// TwinCAT 3 PLC project HMI_PLC
// ProgramVersion: 3.1.4024.0
// libraries:
//   State Machine Twincat, * (Home)
//   Tc2_Standard, * (Beckhoff Automation GmbH)
//   Tc2_System, * (Beckhoff Automation GmbH)
//   Tc3_JsonXml, * (Beckhoff Automation GmbH)
//   Tc3_Module, * (Beckhoff Automation GmbH)
//   VisuSymbols,3.5.10.0,System
// project tree:
//   DUTs/ ST_CameraStates.TcDUT
//   GVLs/ Hardware_Mapping.TcGVL, Cognex_Mapping.TcGVL
//   / PlcTask.TcTTO
//   POUs/ MAIN.TcPOU, _5000_PRG_Aborting.TcPOU, _1000_PRG_Homing.TcPOU, _3000_PRG_Running.TcPOU, _2000_PRG_Stopping.TcPOU, _4000_PRG_Pausing.TcPOU, _6000_PRG_Proceeding.TcPOU, VisualizationManager.TcVMO (not stored)
// real-time tasks:
//   TASK PlcTask: cycle T#10ms, priority 20, ADS port 350
//   TASK VISU_TASK: cycle T#200000us, priority 30, ADS port 351
//   TASK IO Task New: cycle T#1ms, priority 1, ADS port 301
// motion (NC):
//   TASK NC-Task 1 SAF: cycle T#2ms, priority 4, ADS port 501
//   TASK NC-Task 1 SVB: cycle T#10ms, priority 8, ADS port 511
//   AXIS Axis 1 (id 1)
//     OtherSettings: AllowMotionCmdToSlave=true
//     encoder EncType=4
//       EncPara: MaxCount=#x0000ffff
//         Inc: RefSoftSyncMask=#x0000ffff
//     drive DrvType=24
//       Analog: TorqueSetpointScale=10, ScaleFactorActTorque=0.1
//       TimeComp: TaskDelayCycles=1
//     controller CtrType=1
//       CtrPara: PriorControlFactor=1
//         Observer: BandWidth=20
//   AXIS Axis 2 (id 2)
//     OtherSettings: AllowMotionCmdToSlave=true
//     encoder EncType=4
//       EncPara: MaxCount=#x0000ffff
//         Inc: RefSoftSyncMask=#x0000ffff
//     drive DrvType=24
//       Analog: TorqueSetpointScale=10, ScaleFactorActTorque=0.1
//       TimeComp: TaskDelayCycles=1
//     controller CtrType=1
//       CtrPara: PriorControlFactor=1
//         Observer: BandWidth=20
// I/O:
//   DEVICE Device 1 (TC3 EIP Scanner), AmsNetId 172.18.236.100.2.1
//     Box 1 (In-Sight 7000 Series) // <INFO> </INFO> <EDS> C:\TwinCAT\3.1\Config\Io\EtherNetIP\02A6006401090C00.eds </EDS>
//   DEVICE Device 2 (EtherCAT), AmsNetId 172.18.236.100.3.1
//     Term 2 (EK1100) [EK1100 EtherCAT Coupler (2A E-Bus)]
//       Term 3 (EL1008) [EL1008 8Ch. Dig. Input 24V, 3ms]
//       Term 4 (EL1008) [EL1008 8Ch. Dig. Input 24V, 3ms]
//       Term 5 (EL2008) [EL2008 8Ch. Dig. Output 24V, 0.5A]
//       Term 6 (EL2008) [EL2008 8Ch. Dig. Output 24V, 0.5A]
//       Term 7 (EL7047) [EL7047 1Ch. Stepper motor output stage (50V, 5A)]
//       Term 8 (EL7047) [EL7047 1Ch. Stepper motor output stage (50V, 5A)]
//       Term 8 (EL9011) [EL9011 End Terminal]
// variable links:
//   NC-Task 1 SAF/Axes/Axis 1 <-> Device 2 (EtherCAT)/Term 2 (EK1100)/Term 7 (EL7047)
//     Drive/Inputs/In/nState1 @bit 3 <-> STM Status/Status/Error
//     Drive/Inputs/In/nState1 @bit 7 <-> STM Status/Status/Motor stall
//     Drive/Inputs/In/nState1 @bit 5 <-> STM Status/Status/Moving negative
//     Drive/Inputs/In/nState1 @bit 4 <-> STM Status/Status/Moving positive
//     Drive/Inputs/In/nState1 @bit 1 <-> STM Status/Status/Ready
//     Drive/Inputs/In/nState1 <-> STM Status/Status/Ready to enable
//     Drive/Inputs/In/nState1 @bit 6 <-> STM Status/Status/Torque reduced
//     Drive/Inputs/In/nState1 @bit 2 <-> STM Status/Status/Warning
//     Drive/Inputs/In/nState2 @bit 3 <-> STM Status/Status/Digital input 1
//     Drive/Inputs/In/nState2 @bit 4 <-> STM Status/Status/Digital input 2
//     Drive/Inputs/In/nState2 @bit 5 <-> STM Status/Status/Sync error
//     Drive/Inputs/In/nState2 @bit 7 <-> STM Status/Status/TxPDO Toggle
//     Drive/Inputs/In/nState4 @bit 1 <-> WcState/InputToggle
//     Drive/Inputs/In/nState4 <-> WcState/WcState
//     Drive/Outputs/Out/nCtrl1 <-> STM Control/Control/Enable
//     Drive/Outputs/Out/nCtrl1 @bit 2 <-> STM Control/Control/Reduce torque
//     Drive/Outputs/Out/nCtrl1 @bit 1 <-> STM Control/Control/Reset
//     Drive/Outputs/Out/nCtrl2 @bit 3 <-> STM Control/Control/Digital output 1
//     Drive/Outputs/Out/nDataOut2[0] <-> STM Velocity/Velocity
//     Enc/Inputs/In/nDataIn1[0] <-> ENC Status compact/Counter value
//     Enc/Inputs/In/nDataIn2[0] <-> ENC Status compact/Latch value
//     Enc/Inputs/In/nState1 @bit 4 <-> ENC Status compact/Status/Counter overflow
//     Enc/Inputs/In/nState1 @bit 3 <-> ENC Status compact/Status/Counter underflow
//     Enc/Inputs/In/nState1 @bit 7 <-> ENC Status compact/Status/Extrapolation stall
//     Enc/Inputs/In/nState1 <-> ENC Status compact/Status/Latch C valid
//     Enc/Inputs/In/nState1 @bit 1 <-> ENC Status compact/Status/Latch extern valid
//     Enc/Inputs/In/nState1 @bit 2 <-> ENC Status compact/Status/Set counter done
//     Enc/Inputs/In/nState2 @bit 4 <-> ENC Status compact/Status/Status of extern latch
//     Enc/Inputs/In/nState2 <-> ENC Status compact/Status/Status of input A
//     Enc/Inputs/In/nState2 @bit 1 <-> ENC Status compact/Status/Status of input B
//     Enc/Inputs/In/nState2 @bit 2 <-> ENC Status compact/Status/Status of input C
//     Enc/Inputs/In/nState2 @bit 5 <-> ENC Status compact/Status/Sync error
//     Enc/Inputs/In/nState2 @bit 7 <-> ENC Status compact/Status/TxPDO Toggle
//     Enc/Inputs/In/nState4 @bit 1 <-> WcState/InputToggle
//     Enc/Inputs/In/nState4 <-> WcState/WcState
//     Enc/Outputs/Out/nCtrl1 <-> ENC Control compact/Control/Enable latch C
//     Enc/Outputs/Out/nCtrl1 @bit 3 <-> ENC Control compact/Control/Enable latch extern on negative edge
//     Enc/Outputs/Out/nCtrl1 @bit 1 <-> ENC Control compact/Control/Enable latch extern on positive edge
//     Enc/Outputs/Out/nCtrl1 @bit 2 <-> ENC Control compact/Control/Set counter
//     Enc/Outputs/Out/nDataOut1[0] <-> ENC Control compact/Set counter value
//   NC-Task 1 SAF/Axes/Axis 2 <-> Device 2 (EtherCAT)/Term 2 (EK1100)/Term 8 (EL7047)
//     Drive/Inputs/In/nState1 @bit 3 <-> STM Status/Status/Error
//     Drive/Inputs/In/nState1 @bit 7 <-> STM Status/Status/Motor stall
//     Drive/Inputs/In/nState1 @bit 5 <-> STM Status/Status/Moving negative
//     Drive/Inputs/In/nState1 @bit 4 <-> STM Status/Status/Moving positive
//     Drive/Inputs/In/nState1 @bit 1 <-> STM Status/Status/Ready
//     Drive/Inputs/In/nState1 <-> STM Status/Status/Ready to enable
//     Drive/Inputs/In/nState1 @bit 6 <-> STM Status/Status/Torque reduced
//     Drive/Inputs/In/nState1 @bit 2 <-> STM Status/Status/Warning
//     Drive/Inputs/In/nState2 @bit 3 <-> STM Status/Status/Digital input 1
//     Drive/Inputs/In/nState2 @bit 4 <-> STM Status/Status/Digital input 2
//     Drive/Inputs/In/nState2 @bit 5 <-> STM Status/Status/Sync error
//     Drive/Inputs/In/nState2 @bit 7 <-> STM Status/Status/TxPDO Toggle
//     Drive/Inputs/In/nState4 @bit 1 <-> WcState/InputToggle
//     Drive/Inputs/In/nState4 <-> WcState/WcState
//     Drive/Outputs/Out/nCtrl1 <-> STM Control/Control/Enable
//     Drive/Outputs/Out/nCtrl1 @bit 2 <-> STM Control/Control/Reduce torque
//     Drive/Outputs/Out/nCtrl1 @bit 1 <-> STM Control/Control/Reset
//     Drive/Outputs/Out/nCtrl2 @bit 3 <-> STM Control/Control/Digital output 1
//     Drive/Outputs/Out/nDataOut2[0] <-> STM Velocity/Velocity
//     Enc/Inputs/In/nDataIn1[0] <-> ENC Status compact/Counter value
//     Enc/Inputs/In/nDataIn2[0] <-> ENC Status compact/Latch value
//     Enc/Inputs/In/nState1 @bit 4 <-> ENC Status compact/Status/Counter overflow
//     Enc/Inputs/In/nState1 @bit 3 <-> ENC Status compact/Status/Counter underflow
//     Enc/Inputs/In/nState1 @bit 7 <-> ENC Status compact/Status/Extrapolation stall
//     Enc/Inputs/In/nState1 <-> ENC Status compact/Status/Latch C valid
//     Enc/Inputs/In/nState1 @bit 1 <-> ENC Status compact/Status/Latch extern valid
//     Enc/Inputs/In/nState1 @bit 2 <-> ENC Status compact/Status/Set counter done
//     Enc/Inputs/In/nState2 @bit 4 <-> ENC Status compact/Status/Status of extern latch
//     Enc/Inputs/In/nState2 <-> ENC Status compact/Status/Status of input A
//     Enc/Inputs/In/nState2 @bit 1 <-> ENC Status compact/Status/Status of input B
//     Enc/Inputs/In/nState2 @bit 2 <-> ENC Status compact/Status/Status of input C
//     Enc/Inputs/In/nState2 @bit 5 <-> ENC Status compact/Status/Sync error
//     Enc/Inputs/In/nState2 @bit 7 <-> ENC Status compact/Status/TxPDO Toggle
//     Enc/Inputs/In/nState4 @bit 1 <-> WcState/InputToggle
//     Enc/Inputs/In/nState4 <-> WcState/WcState
//     Enc/Outputs/Out/nCtrl1 <-> ENC Control compact/Control/Enable latch C
//     Enc/Outputs/Out/nCtrl1 @bit 3 <-> ENC Control compact/Control/Enable latch extern on negative edge
//     Enc/Outputs/Out/nCtrl1 @bit 1 <-> ENC Control compact/Control/Enable latch extern on positive edge
//     Enc/Outputs/Out/nCtrl1 @bit 2 <-> ENC Control compact/Control/Set counter
//     Enc/Outputs/Out/nDataOut1[0] <-> ENC Control compact/Set counter value
//   HMI-PLC/HMI-PLC Instance <-> Device 1 (TC3 EIP Scanner)/Box 1 (In-Sight 7000 Series)
//     PlcTask Inputs/IO_Mapping.inpAcquiring <-> Connection 1 (Input/Output)/Inputs/Acquiring
//     PlcTask Inputs/IO_Mapping.inpAcquisitionID <-> Connection 1 (Input/Output)/Inputs/Acquisition ID
//     PlcTask Inputs/IO_Mapping.inpCommandComplete <-> Connection 1 (Input/Output)/Inputs/Command Complete
//     PlcTask Inputs/IO_Mapping.inpCommandExecuting <-> Connection 1 (Input/Output)/Inputs/Command Executing
//     PlcTask Inputs/IO_Mapping.inpCommandFailed <-> Connection 1 (Input/Output)/Inputs/Command Failed
//     PlcTask Inputs/IO_Mapping.inpCurrentJobID <-> Connection 1 (Input/Output)/Inputs/Current Job ID
//     PlcTask Inputs/IO_Mapping.inpExposureComplete <-> Connection 1 (Input/Output)/Inputs/Exposure Complete
//     PlcTask Inputs/IO_Mapping.inpInspecting <-> Connection 1 (Input/Output)/Inputs/Inspecting
//     PlcTask Inputs/IO_Mapping.inpInspectionComplete <-> Connection 1 (Input/Output)/Inputs/Inspection Complete
//     PlcTask Inputs/IO_Mapping.inpInspectionID <-> Connection 1 (Input/Output)/Inputs/Inspection ID
//     PlcTask Inputs/IO_Mapping.inpInspectionResultCode <-> Connection 1 (Input/Output)/Inputs/Inspection Result Code
//     PlcTask Inputs/IO_Mapping.inpInspectionResults <-> Connection 1 (Input/Output)/Inputs/Inspection Results
//     PlcTask Inputs/IO_Mapping.inpInspectionResults{1..10} <-> Connection 1 (Input/Output)/Inputs/Inspection Results_{1..10}  (10 links)
//     PlcTask Inputs/IO_Mapping.inpJobPass <-> Connection 1 (Input/Output)/Inputs/Job Pass
//     PlcTask Inputs/IO_Mapping.inpMissedAcq <-> Connection 1 (Input/Output)/Inputs/Missed Acq
//     PlcTask Inputs/IO_Mapping.inpOfflineReason <-> Connection 1 (Input/Output)/Inputs/Offline Reason
//     PlcTask Inputs/IO_Mapping.inpOnline <-> Connection 1 (Input/Output)/Inputs/Online
//     PlcTask Inputs/IO_Mapping.inpResultsBufferOverrun <-> Connection 1 (Input/Output)/Inputs/Results Buffer Overrun
//     PlcTask Inputs/IO_Mapping.inpResultsValid <-> Connection 1 (Input/Output)/Inputs/Results Valid
//     PlcTask Inputs/IO_Mapping.inpTestRunReady <-> Connection 1 (Input/Output)/Inputs/Test Run Ready
//     PlcTask Inputs/IO_Mapping.inpTriggerAck <-> Connection 1 (Input/Output)/Inputs/Trigger Ack
//     PlcTask Inputs/IO_Mapping.inpTriggerReady <-> Connection 1 (Input/Output)/Inputs/Trigger Ready
//     PlcTask Outputs/IO_Mapping.outBufferResultsEnable <-> Connection 1 (Input/Output)/Outputs/Buffer Results Enable
//     PlcTask Outputs/IO_Mapping.outCommand <-> Connection 1 (Input/Output)/Outputs/Command
//     PlcTask Outputs/IO_Mapping.outExecuteCommand <-> Connection 1 (Input/Output)/Outputs/Execute Command
//     PlcTask Outputs/IO_Mapping.outInspectionResultsAck <-> Connection 1 (Input/Output)/Outputs/Inspection Results Ack
//     PlcTask Outputs/IO_Mapping.outSetOffline <-> Connection 1 (Input/Output)/Outputs/Set Offline
//     PlcTask Outputs/IO_Mapping.outSoftEvent{0..7} <-> Connection 1 (Input/Output)/Outputs/Soft Event {0..7}  (8 links)
//     PlcTask Outputs/IO_Mapping.outTriggerCamera <-> Connection 1 (Input/Output)/Outputs/Trigger
//     PlcTask Outputs/IO_Mapping.outTriggerEnable <-> Connection 1 (Input/Output)/Outputs/Trigger Enable
//     PlcTask Outputs/IO_Mapping.outUserData <-> Connection 1 (Input/Output)/Outputs/User Data
//     PlcTask Outputs/IO_Mapping.outUserData{1..10} <-> Connection 1 (Input/Output)/Outputs/User Data_{1..10}  (10 links)
//   HMI-PLC/HMI-PLC Instance <-> Device 2 (EtherCAT)/Term 2 (EK1100)/Term 3 (EL1008)
//     PlcTask Inputs/IO_Mapping.input1 <-> Channel 1/Input
//     PlcTask Inputs/IO_Mapping.input2 <-> Channel 2/Input
//   HMI-PLC/HMI-PLC Instance <-> Device 2 (EtherCAT)/Term 2 (EK1100)/Term 5 (EL2008)
//     PlcTask Outputs/IO_Mapping.output1 <-> Channel 1/Output
//     PlcTask Outputs/IO_Mapping.output2 <-> Channel 2/Output

CONFIGURATION HMI_PLC
    RESOURCE PLC ON TwinCAT3
        TASK PlcTask(INTERVAL := T#10ms, PRIORITY := 20);
        PROGRAM MAIN WITH PlcTask : MAIN;
    END_RESOURCE
END_CONFIGURATION

// ---- DUTs/ST_CameraStates.TcDUT
TYPE ST_CameraState :
STRUCT
    stsIdle              : BOOL := FALSE;
    stsReadyToTrigger    : BOOL := FALSE;
    stsTriggering        : BOOL := FALSE;
    stsAcquiring         : BOOL := FALSE;
    stsWaitResults       : BOOL := FALSE;
    stsProcessResults    : BOOL := FALSE;
    stsError             : BOOL := FALSE;
END_STRUCT
END_TYPE

// ---- GVLs/Hardware_Mapping.TcGVL
{attribute 'qualified_only'}
VAR_GLOBAL
END_VAR

// ---- GVLs/Cognex_Mapping.TcGVL
{attribute 'qualified_only'}
VAR_GLOBAL
	
	// COGNEX INSIGHT 7000 EIP EDS MAPPING
	//--------------------------------------
	// Inputs
	inpTriggerReady AT %I* : BOOL;
	inpTriggerAck AT %I* : BOOL;
	inpAcquiring AT %I* : BOOL;
	inpMissedAcq AT %I* : BOOL;
	inpOfflineReason AT %I* : USINT; // 3 bits represented as USINT (8 bits)
	inpOnline AT %I* : BOOL;
	inpInspecting AT %I* : BOOL;
	inpInspectionComplete AT %I* : BOOL;
	inpResultsBufferOverrun AT %I* : BOOL;
	inpResultsValid AT %I* : BOOL;
	inpCommandExecuting AT %I* : BOOL;
	inpCommandComplete AT %I* : BOOL;
	inpCommandFailed AT %I* : BOOL;
	inpNoname0ArrBIT AT %I* : ARRAY[0..1] OF BOOL;
	inpExposureComplete AT %I* : BOOL;
	inpJobPass AT %I* : BOOL;
	inpTestRunReady AT %I* : BOOL;
	inpNoname1ArrBIT AT %I* : ARRAY[0..1] OF BOOL;
	inpCurrentJobID AT %I* : UINT;
	inpAcquisitionID AT %I* : UINT;
	inpInspectionID AT %I* : UINT;
	inpInspectionResultCode AT %I* : INT;
	inpInspectionResults AT %I* : BYTE;
	inpInspectionResults1 AT %I* : BYTE;
	inpInspectionResults2 AT %I* : BYTE;
	inpInspectionResults3 AT %I* : BYTE;
	inpInspectionResults4 AT %I* : BYTE;
	inpInspectionResults5 AT %I* : BYTE;
	inpInspectionResults6 AT %I* : BYTE;
	inpInspectionResults7 AT %I* : BYTE;
	inpInspectionResults8 AT %I* : BYTE;
	inpInspectionResults9 AT %I* : BYTE;
	inpInspectionResults10 AT %I* : BYTE;
	
	// Outputs
	outTriggerEnable AT %Q* : BOOL;
	outTriggerCamera AT %Q* : BOOL;
	outBufferResultsEnable AT %Q* : BOOL;
	outInspectionResultsAck AT %Q* : BOOL;
	outExecuteCommand AT %Q* : BOOL;
	outNoname0ArrBIT AT %Q* : ARRAY[0..1] OF BOOL;
	outSetOffline AT %Q* : BOOL;
	outSoftEvent0 AT %Q* : BOOL;
	outSoftEvent1 AT %Q* : BOOL;
	outSoftEvent2 AT %Q* : BOOL;
	outSoftEvent3 AT %Q* : BOOL;
	outSoftEvent4 AT %Q* : BOOL;
	outSoftEvent5 AT %Q* : BOOL;
	outSoftEvent6 AT %Q* : BOOL;
	outSoftEvent7 AT %Q* : BOOL;
	outCommand AT %Q* : UINT;
	outUserData AT %Q* : BYTE;
	outUserData1 AT %Q* : BYTE;
	outUserData2 AT %Q* : BYTE;
	outUserData3 AT %Q* : BYTE;
	outUserData4 AT %Q* : BYTE;
	outUserData5 AT %Q* : BYTE;
	outUserData6 AT %Q* : BYTE;
	outUserData7 AT %Q* : BYTE;
	outUserData8 AT %Q* : BYTE;
	outUserData9 AT %Q* : BYTE;
	outUserData10 AT %Q* : BYTE;
	//--------------------------------------
	
	
	// Regular IO 
	input1 AT %I* : BOOL;
	input2 AT %I* : BOOL;
	
	output1 AT %Q* : BOOL;
	output2 AT %Q* : BOOL;

END_VAR

// ---- POUs/MAIN.TcPOU
PROGRAM MAIN
VAR
    // State Machine instance
    fbStateMachine : FB_StateMachine;
    
    // HMI interface for state machine
    stateMachineHMI : SM_HMI;
    
    // Current step for state machine - SHARED between state machine and all step programs
    currentStep : ActiveStep;
    
    // State machine command inputs
    smCommands : ST_SM_Commands;
      
    // Test inputs for permissions
    testAutoIntlk : INT := -1;  // All OK by default (-1 = all bits OK)
    testHomePerm : INT := -1;   // All OK by default
    testStartPerm : INT := -1;  // All OK by default
    testProceedPerm : INT := -1; // All OK by default 

	NextStep: DINT; // Next step to be modified by sequences
	
END_VAR

//=============================================================================
// MAIN PROGRAM - State Machine Implementation with Sequence Programs
//=============================================================================

//=============================================================================
// CENTRALIZED INITIAL STEP SETTING
//=============================================================================
// Initialize sequence when first entering any state (CurrentStep.Step = 0)
IF currentStep.Step = 0 THEN
    IF fbStateMachine.Status.Homing THEN
        NextStep := 1000;  // Start homing sequence
        // Force immediate timer reset on state entry
        smCommands.CompleteState := FALSE;
    ELSIF fbStateMachine.Status.Running THEN
        NextStep := 3000;  // Start running sequence
        smCommands.CompleteState := FALSE;
    ELSIF fbStateMachine.Status.Stopping THEN
        NextStep := 2000;  // Start stopping sequence
        smCommands.CompleteState := FALSE;
    ELSIF fbStateMachine.Status.Aborting THEN
        NextStep := 5000;  // Start aborting sequence
        smCommands.CompleteState := FALSE;
    ELSIF fbStateMachine.Status.Pausing THEN
        NextStep := 4000;  // Start pausing sequence
        smCommands.CompleteState := FALSE;
    ELSIF fbStateMachine.Status.Proceeding THEN
        NextStep := 6000;  // Start proceeding sequence
        smCommands.CompleteState := FALSE;
    ELSE
        // No initial step needed
    END_IF;
END_IF;

// Call state machine BEFORE sequences to ensure timer is updated first
fbStateMachine(
    EnableIn := TRUE,              // Enable the state machine
    cfgAutoRun := TRUE,           // Auto run configuration  
    inpAutoIntlk := testAutoIntlk, // Auto interlocks
    inpHomePerm := testHomePerm,   // Home permissions
    inpStartPerm := testStartPerm, // Start permissions
    inpProceedPerm := testProceedPerm, // Proceed permissions
    NextStep := NextStep,  // Next step from active sequence program
    Commands := smCommands,        // Command inputs
    HMI := stateMachineHMI,        // HMI interface
    CurrentStep := currentStep     // Current step (shared with sequences)
);


//=============================================================================
// ALWAYS CALL ALL SEQUENCE PROGRAMS - AFTER STATE MACHINE
//=============================================================================
// This ensures the timer has been properly updated before sequences evaluate
// Call all sequence programs - FB_SequenceStep logic handles which steps are active
// This ensures all tags update in real-time for better HMI visibility
_1000_PRG_Homing(
    CurrentStep := currentStep,
    StepTimerSeconds := REAL_TO_DINT(fbStateMachine.StepInfo.StepTimerSeconds),
    RetrySignal := fbStateMachine.outRetry,
    StateMachineStatus := fbStateMachine.Status,
    NextStep := NextStep
);

_3000_PRG_Running(
    CurrentStep := currentStep,
    StepTimerSeconds := REAL_TO_DINT(fbStateMachine.StepInfo.StepTimerSeconds),
    RetrySignal := fbStateMachine.outRetry,
    StateMachineStatus := fbStateMachine.Status,
    NextStep := NextStep
);

_2000_PRG_Stopping(
    CurrentStep := currentStep,
    StepTimerSeconds := REAL_TO_DINT(fbStateMachine.StepInfo.StepTimerSeconds),
    RetrySignal := fbStateMachine.outRetry,
    StateMachineStatus := fbStateMachine.Status,
    NextStep := NextStep
);

_5000_PRG_Aborting(
    CurrentStep := currentStep,
    StepTimerSeconds := REAL_TO_DINT(fbStateMachine.StepInfo.StepTimerSeconds),
    RetrySignal := fbStateMachine.outRetry,
    StateMachineStatus := fbStateMachine.Status,
    NextStep := NextStep
);

_4000_PRG_Pausing(
    CurrentStep := currentStep,
    StepTimerSeconds := REAL_TO_DINT(fbStateMachine.StepInfo.StepTimerSeconds),
    RetrySignal := fbStateMachine.outRetry,
    StateMachineStatus := fbStateMachine.Status,
    NextStep := NextStep
);

_6000_PRG_Proceeding(
    CurrentStep := currentStep,
    StepTimerSeconds := REAL_TO_DINT(fbStateMachine.StepInfo.StepTimerSeconds),
    RetrySignal := fbStateMachine.outRetry,
    StateMachineStatus := fbStateMachine.Status,
    NextStep := NextStep
);

END_PROGRAM

// ---- POUs/_1000_PRG_Homing.TcPOU
PROGRAM _1000_PRG_Homing
VAR_IN_OUT
    CurrentStep : ActiveStep;  // Shared step structure with state machine
	NextStep: DINT; // Next step to be modified by sequences
END_VAR

VAR_INPUT
    StepTimerSeconds : DINT;   // Timer value from state machine
    RetrySignal : BOOL;        // Retry signal from state machine
    StateMachineStatus : ST_SM_Status;  // Complete state machine status
END_VAR


VAR
    // Step function blocks for homing sequence
    fbStep1000 : FB_SequenceStep;  // Home Initialize
    fbStep1002 : FB_SequenceStep;  // Home Execute
    
    // Step permissives (simulation for testing)
    step1000Perms : INT := -1;     // All OK for step 1000
    step1002Perms : INT := -1;     // All OK for step 1002
    
END_VAR

//=============================================================================
// PRG_Homing - Handles HOMING state sequence (1000-1999)
//=============================================================================
// Step numbering: 1000, 1002 (even numbers)
// Fault steps: 1001, 1003 (odd numbers, +1 of original)
// NOTE: Initial step setting (CurrentStep.Step = 0) is handled in MAIN program


//=============================================================================
// STEP 1000 - HOME INITIALIZE
//=============================================================================
fbStep1000(
    inpStep := CurrentStep.Step,
    cfgStep := 1000,
    cfgNextStep := 1002,
    inpStepTimerSeconds := StepTimerSeconds,
    inpRetry := RetrySignal,
    inpStepPermissives := step1000Perms,
    cfgStepTimeout := 10,  // 10 second timeout
    inpFaultStep := FALSE,
    ActiveStep := CurrentStep
);

// Step 1000 Active Logic
IF fbStep1000.outStepActive THEN
    // Only simulate permissives if step is active but not advancing
    IF fbStep1000.outNextStep = fbStep1000.cfgStep THEN  // Step is waiting for permissives
        // Permissives simulation - Simulate based on timer
        IF StepTimerSeconds < 3 THEN
            step1000Perms := 16#FFFE;  // Bit 0 not OK (not ready yet)
        ELSE
            step1000Perms := -1;  // All permissives OK after 3 seconds
        END_IF;
    END_IF;
    
    // HMI configuration and actions
    CurrentStep.PermsHMI.Name := 'Home Initialize';
    CurrentStep.PermsHMI.Desc[0] := 'System Ready';
    CurrentStep.PermsHMI.Desc[1] := 'Home Position Clear';
    CurrentStep.PermsHMI.Desc[2] := 'Safety Systems OK';
    
    // Add any step-specific actions here
    // Example: Reset position counters, check home sensors, etc.
    
    // FB_SequenceStep determines next step automatically based on permissives
    NextStep := fbStep1000.outNextStep;
ELSE
    // Reset permissives when step is not active (ensures fresh start next time)
    step1000Perms := 16#FFFE;  // Reset to NOT OK when leaving step
END_IF;

//=============================================================================
// STEP 1002 - HOME EXECUTE
//=============================================================================
fbStep1002(
    inpStep := CurrentStep.Step,
    cfgStep := 1002,
    cfgNextStep := 0,  // sequence complete
    inpStepTimerSeconds := StepTimerSeconds,
    inpRetry := RetrySignal,
    inpStepPermissives := step1002Perms,
    cfgStepTimeout := 15,  // 15 second timeout
    inpFaultStep := FALSE,
    ActiveStep := CurrentStep
);

// Step 1002 Active Logic
IF fbStep1002.outStepActive THEN
    // Only simulate permissives if step is active but not advancing
    IF fbStep1002.outNextStep = fbStep1002.cfgStep THEN  // Step is waiting for permissives
        // Permissives simulation - Simulate based on timer
        IF StepTimerSeconds < 8 THEN
            step1002Perms := 16#FFFD;  // Bit 1 not OK (homing not complete)
        ELSE
            step1002Perms := -1;  // All permissives OK after 8 seconds
        END_IF;
    END_IF;
    
    // HMI configuration and actions
    CurrentStep.PermsHMI.Name := 'Home Execute';
    CurrentStep.PermsHMI.Desc[0] := 'Motors Enabled';
    CurrentStep.PermsHMI.Desc[1] := 'Home Sensors Active';
    CurrentStep.PermsHMI.Desc[2] := 'No Emergency Stops';
    
    // Add any step-specific actions here
    // Example: Start homing motion, monitor position feedback, etc.
    
    // FB_SequenceStep determines next step automatically based on permissives
    NextStep := fbStep1002.outNextStep;
ELSE
    // Reset permissives when step is not active (ensures fresh start next time)
    step1002Perms := 16#FFFD;  // Reset to NOT OK when leaving step
END_IF;

END_PROGRAM

// ---- POUs/_3000_PRG_Running.TcPOU
PROGRAM _3000_PRG_Running
VAR_IN_OUT
    CurrentStep : ActiveStep;  // Shared step structure with state machine
	NextStep: DINT; // Next step to be modified by sequences
END_VAR
VAR_INPUT
    StepTimerSeconds : DINT;   // Timer value from state machine
    RetrySignal : BOOL;        // Retry signal from state machine
    StateMachineStatus : ST_SM_Status;  // Complete state machine status
END_VAR

VAR
    // Step function blocks for running sequence
    fbStep3000 : FB_SequenceStep;  // Production Start
    fbStep3002 : FB_SequenceStep;  // Production Execute
    fbStep3004 : FB_SequenceStep;  // Production Quality Check
    fbStep3006 : FB_SequenceStep;  // Packaging Prepare
    fbStep3008 : FB_SequenceStep;  // Production Finalize
    
    // Step permissives (simulation for testing)
    step3000Perms : INT := -1;     // All OK for step 3000
    step3002Perms : INT := -1;     // All OK for step 3002
    step3004Perms : INT := -1;     // All OK for step 3004
    step3006Perms : INT := -1;     // All OK for step 3006
    step3008Perms : INT := -1;     // All OK for step 3008
    
END_VAR

//=============================================================================
// PRG_Running - Handles RUNNING state sequence (3000-3999)
//=============================================================================
// Step numbering: 3000, 3002 (even numbers)
// Fault steps: 3001, 3003 (odd numbers, +1 of original)
// NOTE: Initial step setting (CurrentStep.Step = 0) is handled in MAIN program


//=============================================================================
// STEP 3000 - PRODUCTION START
//=============================================================================
fbStep3000(
    inpStep := CurrentStep.Step,
    cfgStep := 3000,
    cfgNextStep := 3002,
    inpStepTimerSeconds := StepTimerSeconds,
    inpRetry := RetrySignal,
    inpStepPermissives := step3000Perms,
    cfgStepTimeout := 12,  // 12 second timeout
    inpFaultStep := FALSE,
    ActiveStep := CurrentStep
);

// Step 3000 Active Logic
IF fbStep3000.outStepActive THEN
    // Only simulate permissives if step is active but not advancing
    IF fbStep3000.outNextStep = fbStep3000.cfgStep THEN  // Step is waiting for permissives
        // Permissives simulation - Simulate based on timer
        IF StepTimerSeconds < 3 THEN
            step3000Perms := 16#FFFE;  // Bit 0 not OK (not ready yet)
        ELSE
            step3000Perms := -1;  // All permissives OK after 5 seconds
        END_IF;
    END_IF;
    
    // HMI configuration and actions
    CurrentStep.PermsHMI.Name := 'Production Start';
    CurrentStep.PermsHMI.Desc[0] := 'Raw Material Available';
    CurrentStep.PermsHMI.Desc[1] := 'Process Temperature OK';
    CurrentStep.PermsHMI.Desc[2] := 'Quality System Ready';
    
    // Add any step-specific actions here
    // Example: Start production line, initialize process parameters, etc.
    
    // FB_SequenceStep determines next step automatically based on permissives
    NextStep := fbStep3000.outNextStep;
ELSE
    // Reset permissives when step is not active (ensures fresh start next time)
    step3000Perms := 16#FFFE;  // Reset to NOT OK when leaving step
END_IF;

//=============================================================================
// STEP 3002 - PRODUCTION EXECUTE
//=============================================================================
fbStep3002(
    inpStep := CurrentStep.Step,
    cfgStep := 3002,
    cfgNextStep := 3004,
    inpStepTimerSeconds := StepTimerSeconds,
    inpRetry := RetrySignal,
    inpStepPermissives := step3002Perms,
    cfgStepTimeout := 20,  // 20 second timeout
    inpFaultStep := FALSE,
    ActiveStep := CurrentStep
);

// Step 3002 Active Logic
IF fbStep3002.outStepActive THEN
    // Only simulate permissives if step is active but not advancing
    IF fbStep3002.outNextStep = fbStep3002.cfgStep THEN  // Step is waiting for permissives
        // Permissives simulation - Simulate based on timer
        IF StepTimerSeconds < 4 THEN
            step3002Perms := 16#FFFD;  // Bit 1 not OK (production not complete)
        ELSE
            step3002Perms := -1;  // All permissives OK after 15 seconds
        END_IF;
    END_IF;
    
    // HMI configuration and actions
    CurrentStep.PermsHMI.Name := 'Production Execute';
    CurrentStep.PermsHMI.Desc[0] := 'Production Line Running';
    CurrentStep.PermsHMI.Desc[1] := 'Quality Checks Passing';
    CurrentStep.PermsHMI.Desc[2] := 'Output Quality OK';
    
    // Add any step-specific actions here
    // Example: Monitor production process, quality checks, output control, etc.
    
    // FB_SequenceStep determines next step automatically based on permissives
    NextStep := fbStep3002.outNextStep;
ELSE
    // Reset permissives when step is not active (ensures fresh start next time)
    step3002Perms := 16#FFFD;  // Reset to NOT OK when leaving step
END_IF;

//=============================================================================
// STEP 3004 - PRODUCTION QUALITY CHECK
//=============================================================================
fbStep3004(
    inpStep := CurrentStep.Step,
    cfgStep := 3004,
    cfgNextStep := 3006,
    inpStepTimerSeconds := StepTimerSeconds,
    inpRetry := RetrySignal,
    inpStepPermissives := step3004Perms,
    cfgStepTimeout := 12,  // 12 second timeout
    inpFaultStep := FALSE,
    ActiveStep := CurrentStep
);

IF fbStep3004.outStepActive THEN
    // Only simulate permissives if step is active but not advancing
    IF fbStep3004.outNextStep = fbStep3004.cfgStep THEN  // Step is waiting for permissives
        // Simulate based on timer: delay bit 2
        IF StepTimerSeconds < 3 THEN
            step3004Perms := 16#FFFB;  // Bit 2 not OK
        ELSE
            step3004Perms := -1;       // All OK
        END_IF;
    END_IF;

    // HMI configuration and actions
    CurrentStep.PermsHMI.Name := 'Production Quality Check';
    CurrentStep.PermsHMI.Desc[0] := 'Inspection Running';
    CurrentStep.PermsHMI.Desc[1] := 'Reject Bin Clear';
    CurrentStep.PermsHMI.Desc[2] := 'Measurements In Spec';

    // Advance handled by FB
    NextStep := fbStep3004.outNextStep;
ELSE
    step3004Perms := 16#FFFB;  // Reset to NOT OK when leaving step
END_IF;

//=============================================================================
// STEP 3006 - PACKAGING PREPARE
//=============================================================================
fbStep3006(
    inpStep := CurrentStep.Step,
    cfgStep := 3006,
    cfgNextStep := 3008,
    inpStepTimerSeconds := StepTimerSeconds,
    inpRetry := RetrySignal,
    inpStepPermissives := step3006Perms,
    cfgStepTimeout := 15,  // 15 second timeout
    inpFaultStep := FALSE,
    ActiveStep := CurrentStep
);

IF fbStep3006.outStepActive THEN
    // Only simulate permissives if step is active but not advancing
    IF fbStep3006.outNextStep = fbStep3006.cfgStep THEN  // Step is waiting for permissives
        // Simulate based on timer: delay bit 3
        IF StepTimerSeconds < 3 THEN
            step3006Perms := 16#FFF7;  // Bit 3 not OK
        ELSE
            step3006Perms := -1;       // All OK
        END_IF;
    END_IF;

    // HMI configuration and actions
    CurrentStep.PermsHMI.Name := 'Packaging Prepare';
    CurrentStep.PermsHMI.Desc[0] := 'Empty Boxes Available';
    CurrentStep.PermsHMI.Desc[1] := 'Labeler Ready';
    CurrentStep.PermsHMI.Desc[2] := 'Conveyor Clear';

    // Advance handled by FB
    NextStep := fbStep3006.outNextStep;
ELSE
    step3006Perms := 16#FFF7;  // Reset to NOT OK when leaving step
END_IF;

//=============================================================================
// STEP 3008 - PRODUCTION FINALIZE
//=============================================================================
fbStep3008(
    inpStep := CurrentStep.Step,
    cfgStep := 3008,
    cfgNextStep := 0,  // sequence complete
    inpStepTimerSeconds := StepTimerSeconds,
    inpRetry := RetrySignal,
    inpStepPermissives := step3008Perms,
    cfgStepTimeout := 10,  // 10 second timeout
    inpFaultStep := FALSE,
    ActiveStep := CurrentStep
);

IF fbStep3008.outStepActive THEN
    // Only simulate permissives if step is active but not advancing
    IF fbStep3008.outNextStep = fbStep3008.cfgStep THEN  // Step is waiting for permissives
        // Simulate based on timer: delay bit 4
        IF StepTimerSeconds < 4 THEN
            step3008Perms := 16#FFEF;  // Bit 4 not OK
        ELSE
            step3008Perms := -1;       // All OK
        END_IF;
    END_IF;

    // HMI configuration and actions
    CurrentStep.PermsHMI.Name := 'Production Finalize';
    CurrentStep.PermsHMI.Desc[0] := 'Batch Closed';
    CurrentStep.PermsHMI.Desc[1] := 'Reports Generated';
    CurrentStep.PermsHMI.Desc[2] := 'Area Clear';

    // Advance handled by FB
    NextStep := fbStep3008.outNextStep;
ELSE
    step3008Perms := 16#FFEF;  // Reset to NOT OK when leaving step
END_IF;

END_PROGRAM

// ---- POUs/_2000_PRG_Stopping.TcPOU
PROGRAM _2000_PRG_Stopping
VAR_IN_OUT
    CurrentStep : ActiveStep;  // Shared step structure with state machine
	NextStep: DINT; // Next step to be modified by sequences
END_VAR

VAR_INPUT
    StepTimerSeconds : DINT;   // Timer value from state machine
    RetrySignal : BOOL;        // Retry signal from state machine
    StateMachineStatus : ST_SM_Status;  // Complete state machine status
END_VAR

VAR
    // Step function blocks for stopping sequence
    fbStep2000 : FB_SequenceStep;  // Stop Prepare
    fbStep2002 : FB_SequenceStep;  // Stop Execute
    
    // Step permissives (simulation for testing)
    step2000Perms : INT := -1;     // All OK for step 2000
    step2002Perms : INT := -1;     // All OK for step 2002
    
END_VAR

//=============================================================================
// PRG_Stopping - Handles STOPPING state sequence (2000-2999)
//=============================================================================
// Step numbering: 2000, 2002 (even numbers)
// Fault steps: 2001, 2003 (odd numbers, +1 of original)
// NOTE: Initial step setting (CurrentStep.Step = 0) is handled in MAIN program


//=============================================================================
// STEP 2000 - STOP PREPARE
//=============================================================================
fbStep2000(
    inpStep := CurrentStep.Step,
    cfgStep := 2000,
    cfgNextStep := 2002,
    inpStepTimerSeconds := StepTimerSeconds,
    inpRetry := RetrySignal,
    inpStepPermissives := step2000Perms,
    cfgStepTimeout := 8,  // 8 second timeout
    inpFaultStep := FALSE,
    ActiveStep := CurrentStep
);

// Step 2000 Active Logic
IF fbStep2000.outStepActive THEN
    // Only simulate permissives if step is active but not advancing
    IF fbStep2000.outNextStep = fbStep2000.cfgStep THEN  // Step is waiting for permissives
        // Permissives simulation - Simulate based on timer
        IF StepTimerSeconds < 4 THEN
            step2000Perms := 16#FFFE;  // Bit 0 not OK (not ready yet)
        ELSE
            step2000Perms := -1;  // All permissives OK after 4 seconds
        END_IF;
    END_IF;
    
    // HMI configuration and actions
    CurrentStep.PermsHMI.Name := 'Stop Prepare';
    CurrentStep.PermsHMI.Desc[0] := 'Production Safe to Stop';
    CurrentStep.PermsHMI.Desc[1] := 'Work in Progress Clear';
    CurrentStep.PermsHMI.Desc[2] := 'Equipment Ready for Stop';
    
    // Add any step-specific actions here
    // Example: Complete current work cycle, prepare for safe stop, etc.
    
    // FB_SequenceStep determines next step automatically based on permissives
    NextStep := fbStep2000.outNextStep;
ELSE
    // Reset permissives when step is not active (ensures fresh start next time)
    step2000Perms := 16#FFFE;  // Reset to NOT OK when leaving step
END_IF;

//=============================================================================
// STEP 2002 - STOP EXECUTE
//=============================================================================
fbStep2002(
    inpStep := CurrentStep.Step,
    cfgStep := 2002,
    cfgNextStep := 0,  // sequence complete
    inpStepTimerSeconds := StepTimerSeconds,
    inpRetry := RetrySignal,
    inpStepPermissives := step2002Perms,
    cfgStepTimeout := 12,  // 12 second timeout
    inpFaultStep := FALSE,
    ActiveStep := CurrentStep
);

// Step 2002 Active Logic
IF fbStep2002.outStepActive THEN
    // Only simulate permissives if step is active but not advancing
    IF fbStep2002.outNextStep = fbStep2002.cfgStep THEN  // Step is waiting for permissives
        // Permissives simulation - Simulate based on timer
        IF StepTimerSeconds < 8 THEN
            step2002Perms := 16#FFFD;  // Bit 1 not OK (stop not complete)
        ELSE
            step2002Perms := -1;  // All permissives OK after 8 seconds
        END_IF;
    END_IF;
    
    // HMI configuration and actions
    CurrentStep.PermsHMI.Name := 'Stop Execute';
    CurrentStep.PermsHMI.Desc[0] := 'Motors Stopping';
    CurrentStep.PermsHMI.Desc[1] := 'Systems Powering Down';
    CurrentStep.PermsHMI.Desc[2] := 'Safe State Achieved';
    
    // Add any step-specific actions here
    // Example: Stop motors, power down systems, secure valves, etc.
    
    // FB_SequenceStep determines next step automatically based on permissives
    NextStep := fbStep2002.outNextStep;
ELSE
    // Reset permissives when step is not active (ensures fresh start next time)
    step2002Perms := 16#FFFD;  // Reset to NOT OK when leaving step
END_IF;

END_PROGRAM

// ---- POUs/_5000_PRG_Aborting.TcPOU
PROGRAM _5000_PRG_Aborting
VAR_IN_OUT
    CurrentStep : ActiveStep;  // Shared step structure with state machine
	NextStep: DINT; // Next step to be modified by sequences
END_VAR

VAR_INPUT
    StepTimerSeconds : DINT;   // Timer value from state machine
    RetrySignal : BOOL;        // Retry signal from state machine
    StateMachineStatus : ST_SM_Status;  // Complete state machine status
END_VAR

VAR
    // Step function blocks for aborting sequence
    fbStep5000 : FB_SequenceStep;  // Abort Prepare
    fbStep5002 : FB_SequenceStep;  // Abort Execute
    
    // Step permissives (simulation for testing)
    step5000Perms : INT := -1;     // All OK for step 5000
    step5002Perms : INT := -1;     // All OK for step 5002
    
END_VAR

//=============================================================================
// PRG_Aborting - Handles ABORTING state sequence (5000-5999)
//=============================================================================
// Step numbering: 5000, 5002 (even numbers)
// Fault steps: 5001, 5003 (odd numbers, +1 of original)
// NOTE: Initial step setting (CurrentStep.Step = 0) is handled in MAIN program



//=============================================================================
// STEP 5000 - ABORT PREPARE
//=============================================================================
fbStep5000(
    inpStep := CurrentStep.Step,
    cfgStep := 5000,
    cfgNextStep := 5002,
    inpStepTimerSeconds := StepTimerSeconds,
    inpRetry := RetrySignal,
    inpStepPermissives := step5000Perms,
    cfgStepTimeout := 5,  // 5 second timeout (quick abort)
    inpFaultStep := FALSE,
    ActiveStep := CurrentStep
);

// Step 5000 Active Logic
IF fbStep5000.outStepActive THEN
    // Only simulate permissives if step is active but not advancing
    IF fbStep5000.outNextStep = fbStep5000.cfgStep THEN  // Step is waiting for permissives
        // Permissives simulation - Simulate based on timer
        IF StepTimerSeconds < 2 THEN
            step5000Perms := 16#FFFE;  // Bit 0 not OK (not ready yet)
        ELSE
            step5000Perms := -1;  // All permissives OK after 2 seconds
        END_IF;
    END_IF;
    
    // HMI configuration and actions
    CurrentStep.PermsHMI.Name := 'Abort Prepare';
    CurrentStep.PermsHMI.Desc[0] := 'Emergency Stop Clear';
    CurrentStep.PermsHMI.Desc[1] := 'Safety Systems Active';
    CurrentStep.PermsHMI.Desc[2] := 'Personnel Clear';
    
    // Add any step-specific actions here
    // Example: Set emergency stop relays, activate warning lights, etc.
    
    // FB_SequenceStep determines next step automatically based on permissives
    NextStep := fbStep5000.outNextStep;
ELSE
    // Reset permissives when step is not active (ensures fresh start next time)
    step5000Perms := 16#FFFE;  // Reset to NOT OK when leaving step
END_IF;

//=============================================================================
// STEP 5002 - ABORT EXECUTE  
//=============================================================================
fbStep5002(
    inpStep := CurrentStep.Step,
    cfgStep := 5002,
    cfgNextStep := 0,  // sequence complete
    inpStepTimerSeconds := StepTimerSeconds,
    inpRetry := RetrySignal,
    inpStepPermissives := step5002Perms,
    cfgStepTimeout := 10,  // 10 second timeout
    inpFaultStep := FALSE,
    ActiveStep := CurrentStep
);

// Step 5002 Active Logic
IF fbStep5002.outStepActive THEN
    // Only simulate permissives if step is active but not advancing
    IF fbStep5002.outNextStep = fbStep5002.cfgStep THEN  // Step is waiting for permissives
        // Permissives simulation - Simulate based on timer
        IF StepTimerSeconds < 6 THEN
            step5002Perms := 16#FFFD;  // Bit 1 not OK (abort not complete)
        ELSE
            step5002Perms := -1;  // All permissives OK after 6 seconds
        END_IF;
    END_IF;
    
    // HMI configuration and actions
    CurrentStep.PermsHMI.Name := 'Abort Execute';
    CurrentStep.PermsHMI.Desc[0] := 'Emergency Shutdown Active';
    CurrentStep.PermsHMI.Desc[1] := 'Systems Securing';
    CurrentStep.PermsHMI.Desc[2] := 'Safe State Reached';
    
    // Add any step-specific actions here
    // Example: Execute shutdown sequence, secure valves, stop motors, etc.
    
    // FB_SequenceStep determines next step automatically based on permissives
     NextStep := fbStep5002.outNextStep;
ELSE
    // Reset permissives when step is not active (ensures fresh start next time)
    step5002Perms := 16#FFFD;  // Reset to NOT OK when leaving step
END_IF;

END_PROGRAM

// ---- POUs/_4000_PRG_Pausing.TcPOU
PROGRAM _4000_PRG_Pausing
VAR_IN_OUT
    CurrentStep : ActiveStep;
    NextStep    : DINT;
END_VAR
VAR_INPUT
    StepTimerSeconds   : DINT;
    RetrySignal        : BOOL;
    StateMachineStatus : ST_SM_Status;
END_VAR
VAR
    fbStep4000 : FB_SequenceStep; // Pausing prepare
    fbStep4002 : FB_SequenceStep; // Pausing execute
    step4000Perms : INT := -1;
    step4002Perms : INT := -1;
END_VAR


// STEP 4000 - PAUSING PREPARE
fbStep4000(
    inpStep := CurrentStep.Step,
    cfgStep := 4000,
    cfgNextStep := 4002,
    inpStepTimerSeconds := StepTimerSeconds,
    inpRetry := RetrySignal,
    inpStepPermissives := step4000Perms,
    cfgStepTimeout := 5,
    inpFaultStep := FALSE,
    ActiveStep := CurrentStep
);
IF fbStep4000.outStepActive THEN
    IF fbStep4000.outNextStep = fbStep4000.cfgStep THEN
        IF StepTimerSeconds < 2 THEN
            step4000Perms := 16#FFFE;
        ELSE
            step4000Perms := -1;
        END_IF;
    END_IF;
    CurrentStep.PermsHMI.Name := 'Pausing Prepare';
    CurrentStep.PermsHMI.Desc[0] := 'Prepare to Pause';
    CurrentStep.PermsHMI.Desc[1] := 'Buffer Operations';
    CurrentStep.PermsHMI.Desc[2] := 'Safe To Pause';
    NextStep := fbStep4000.outNextStep;
ELSE
    step4000Perms := 16#FFFE;
END_IF;

// STEP 4002 - PAUSING EXECUTE
fbStep4002(
    inpStep := CurrentStep.Step,
    cfgStep := 4002,
    cfgNextStep := 0, // sequence complete
    inpStepTimerSeconds := StepTimerSeconds,
    inpRetry := RetrySignal,
    inpStepPermissives := step4002Perms,
    cfgStepTimeout := 8,
    inpFaultStep := FALSE,
    ActiveStep := CurrentStep
);
IF fbStep4002.outStepActive THEN
    IF fbStep4002.outNextStep = fbStep4002.cfgStep THEN
        IF StepTimerSeconds < 5 THEN
            step4002Perms := 16#FFFD;
        ELSE
            step4002Perms := -1;
        END_IF;
    END_IF;
    CurrentStep.PermsHMI.Name := 'Pausing Execute';
    CurrentStep.PermsHMI.Desc[0] := 'Pausing';
    CurrentStep.PermsHMI.Desc[1] := 'Drive/Actuator Hold';
    CurrentStep.PermsHMI.Desc[2] := 'Safe State';
    NextStep := fbStep4002.outNextStep;
ELSE
    step4002Perms := 16#FFFD;
END_IF;

END_PROGRAM

// ---- POUs/_6000_PRG_Proceeding.TcPOU
PROGRAM _6000_PRG_Proceeding
VAR_IN_OUT
    CurrentStep : ActiveStep;
    NextStep    : DINT;
END_VAR
VAR_INPUT
    StepTimerSeconds   : DINT;
    RetrySignal        : BOOL;
    StateMachineStatus : ST_SM_Status;
END_VAR
VAR
    fbStep6000 : FB_SequenceStep; // Proceeding prepare
    fbStep6002 : FB_SequenceStep; // Proceeding resume
    step6000Perms : INT := -1;
    step6002Perms : INT := -1;
END_VAR


// STEP 6000 - PROCEEDING PREPARE
fbStep6000(
    inpStep := CurrentStep.Step,
    cfgStep := 6000,
    cfgNextStep := 6002,
    inpStepTimerSeconds := StepTimerSeconds,
    inpRetry := RetrySignal,
    inpStepPermissives := step6000Perms,
    cfgStepTimeout := 5,
    inpFaultStep := FALSE,
    ActiveStep := CurrentStep
);
IF fbStep6000.outStepActive THEN
    IF fbStep6000.outNextStep = fbStep6000.cfgStep THEN
        IF StepTimerSeconds < 2 THEN
            step6000Perms := 16#FFFE;
        ELSE
            step6000Perms := -1;
        END_IF;
    END_IF;
    CurrentStep.PermsHMI.Name := 'Proceed Prepare';
    CurrentStep.PermsHMI.Desc[0] := 'Ready to Resume';
    CurrentStep.PermsHMI.Desc[1] := 'Interlocks OK';
    CurrentStep.PermsHMI.Desc[2] := 'Resources Available';
    NextStep := fbStep6000.outNextStep;
ELSE
    step6000Perms := 16#FFFE;
END_IF;

// STEP 6002 - PROCEEDING RESUME
fbStep6002(
    inpStep := CurrentStep.Step,
    cfgStep := 6002,
    cfgNextStep := 0, // sequence complete
    inpStepTimerSeconds := StepTimerSeconds,
    inpRetry := RetrySignal,
    inpStepPermissives := step6002Perms,
    cfgStepTimeout := 8,
    inpFaultStep := FALSE,
    ActiveStep := CurrentStep
);
IF fbStep6002.outStepActive THEN
    IF fbStep6002.outNextStep = fbStep6002.cfgStep THEN
        IF StepTimerSeconds < 4 THEN
            step6002Perms := 16#FFFD;
        ELSE
            step6002Perms := -1;
        END_IF;
    END_IF;
    CurrentStep.PermsHMI.Name := 'Proceed Resume';
    CurrentStep.PermsHMI.Desc[0] := 'Resuming';
    CurrentStep.PermsHMI.Desc[1] := 'Synchronizing';
    CurrentStep.PermsHMI.Desc[2] := 'Back to Operation';
    NextStep := fbStep6002.outNextStep;
ELSE
    step6002Perms := 16#FFFD;
END_IF;

END_PROGRAM
